PROGRAM P5_05_Screenshot
VAR
		fbScreenshot					:NT_StartProcess;
		tonDisable						:TON;
		bDisable						:BOOL;
END_VAR

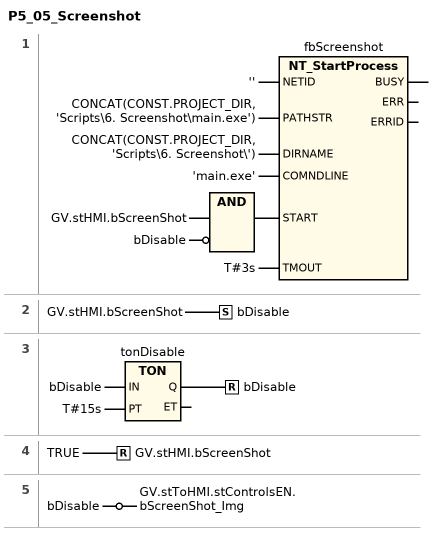
// NETWORK 1
fbScreenshot(
    NETID := '',
    PATHSTR := CONCAT(CONST.PROJECT_DIR,'Scripts\6. Screenshot\main.exe'),
    DIRNAME := CONCAT(CONST.PROJECT_DIR,'Scripts\6. Screenshot\'),
    COMNDLINE := 'main.exe',
    START := GV.stHMI.bScreenShot AND NOT bDisable,
    TMOUT := T#3s); // NT_StartProcess

// NETWORK 2
bDisable S= GV.stHMI.bScreenShot;

// NETWORK 3
tonDisable(IN := bDisable, PT := T#15s); // TON
bDisable R= tonDisable.Q;

// NETWORK 4
GV.stHMI.bScreenShot R= TRUE;

// NETWORK 5
GV.stToHMI.stControlsEN.bScreenShot_Img := NOT bDisable;

END_PROGRAM

(* stored: Version 1.1.0.1, ProductVersion 3.1.4024.12
   POU P5_05_Screenshot: Id {057aadf9-a323-4a87-9f33-6043c9bc93ca}, SpecialFunc None *)
